SUBAPPLICATION MechatronicArm (* Subapplication Type *)
  (* Standard: 61499-2 *)
  (* Version 1.0, 2025-03-21, AK123700 *)
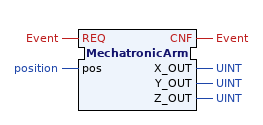
  EVENT_INPUT
    REQ; (* Normal Execution Request *)
  END_EVENT
  EVENT_OUTPUT
    CNF; (* Execution Confirmation *)
  END_EVENT
  VAR_INPUT
    pos : position;
  END_VAR
  VAR_OUTPUT
    X_OUT : UINT;
    Y_OUT : UINT;
    Z_OUT : UINT;
  END_VAR
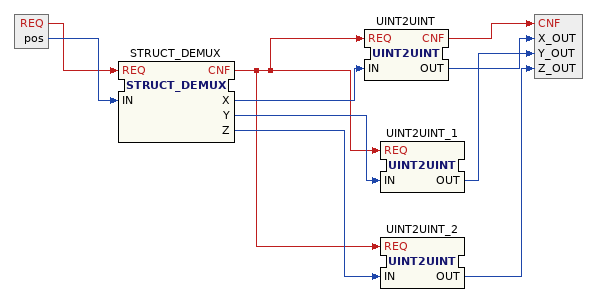
  FBS
    STRUCT_DEMUX : STRUCT_DEMUX; {SET_ATTRIBUTE(StructuredType, position)}
    UINT2UINT_2 : UINT2UINT;
    UINT2UINT_1 : UINT2UINT;
    UINT2UINT : UINT2UINT;
  END_FBS
  EVENT_CONNECTIONS
    REQ TO STRUCT_DEMUX.REQ;
    STRUCT_DEMUX.CNF TO UINT2UINT_2.REQ;
    STRUCT_DEMUX.CNF TO UINT2UINT_1.REQ;
    STRUCT_DEMUX.CNF TO UINT2UINT.REQ;
    UINT2UINT.CNF TO CNF;
  END_CONNECTIONS
  DATA_CONNECTIONS
    pos TO STRUCT_DEMUX.IN;
    UINT2UINT_2.OUT TO Z_OUT;
    UINT2UINT_1.OUT TO Y_OUT;
    UINT2UINT.OUT TO X_OUT;
    STRUCT_DEMUX.X TO UINT2UINT.IN;
    STRUCT_DEMUX.Y TO UINT2UINT_1.IN;
    STRUCT_DEMUX.Z TO UINT2UINT_2.IN;
  END_CONNECTIONS
END_SUBAPPLICATION
